Staubli VAL3: Control_Preset.pgx

public program Control_Preset(num& x_nPreset[] (dimensions=2), num x_nIndex)
  local string l_sItem[5]
  local num l_nNum
  local num l_nKey
  local num l_nData[5]
  local num l_nSelectIndex
begin

  //修改点位的 joint

  for l_nNum=0 to 4
    l_nData[l_nNum]=x_nPreset[x_nIndex,l_nNum]
  endFor



  l_sItem[0]="激光功率  :"+toString("",l_nData[0])
  l_sItem[1]="气体压力  :"+toString("",l_nData[1])
  l_sItem[2]="占空比频率:"+toString("",l_nData[2])
  l_sItem[3]="激光占空比:"+toString("",l_nData[3])
  l_sItem[4]="随动高度  :"+toString("",l_nData[4])

  call Control_BottomS(",,,,,,取消,确定")
  call Control_PanelXY(8,0,15,5)
  call Control_Panel("工艺值")
  call Control_List(l_sItem,l_nSelectIndex)
  while true
    l_nKey=getKey()

    switch l_nKey
      case 261
        l_nSelectIndex=max(0,l_nSelectIndex-1)
      break

      case 266
        l_nSelectIndex=min(l_nSelectIndex+1,5)
      break

      case 278
        for l_nNum=0 to 4
          x_nPreset[x_nIndex,l_nNum]=min(max(l_nData[l_nNum],0),100)
        endFor
        return
      break


      case 277
        return
      break

      case 270
        call Float_Edit(l_nData[l_nSelectIndex],nPanelLTopX+12,l_nSelectIndex+nPanelLTopY+1)
        l_nData[l_nSelectIndex]=min(max(l_nData[l_nSelectIndex],0),100)
      break

    endSwitch

    if l_nKey!=-1

      l_sItem[0]="激光功率  :"+toString("",l_nData[0])
      l_sItem[1]="气体压力  :"+toString("",l_nData[1])
      l_sItem[2]="占空比频率:"+toString("",l_nData[2])
      l_sItem[3]="激光占空比:"+toString("",l_nData[3])
      l_sItem[4]="随动高度  :"+toString("",l_nData[4])
      call Control_List(l_sItem,l_nSelectIndex)

    endIf






  endWhile





end
